INTERFACE I_State

PROPERTY Description : STRING
GET
END_GET
END_PROPERTY

METHOD ErrorDetected : BOOL
VAR_IN_OUT
	errorEvents		: ST_ErrorEvents;
END_VAR
END_METHOD

METHOD HeatIsRequested : BOOL
VAR_INPUT
END_VAR
END_METHOD

METHOD LimitValuesAreExceeded  : BOOL
VAR_INPUT
END_VAR
END_METHOD

PROPERTY Name : String
GET
END_GET
END_PROPERTY

PROPERTY State : E_State
GET
END_GET
END_PROPERTY

METHOD TargetTemperatureReached : BOOL
VAR_INPUT
END_VAR
END_METHOD

METHOD UserPressedConfirmationButton : BOOL
VAR_INPUT
END_VAR
END_METHOD

METHOD UserPressedSwitchOffButton : BOOL
VAR_INPUT
END_VAR
END_METHOD

METHOD UserPressedSwitchOnButton : BOOL
VAR_INPUT
END_VAR
END_METHOD

METHOD WaterHasCooledDown : BOOL
VAR_INPUT
END_VAR
END_METHOD

END_INTERFACE

(* stored: Version 1.1.0.1
   Itf I_State: Id {ebee4276-c4cf-4931-866b-4251da6de24d}
   Property Description: Id {09fe3b11-4466-4002-a19f-d7f98022308d}
   Get Get: Id {fb376b64-5463-4c2d-a1bb-8dc6a8df688f}
   Method ErrorDetected: Id {1fadc6df-44ce-4163-8a9d-0b84f9d6da56}
   Method HeatIsRequested: Id {bd7aa1f8-5748-4535-ba75-c3d1e68d26b3}
   Method LimitValuesAreExceeded: Id {00119294-6b09-4037-a5f2-bdd6e49bdada}
   Property Name: Id {185febd2-623d-4463-8457-cd856daf23b0}
   Get Get: Id {706e1d71-bb03-45f8-9d3a-58a361b141c0}
   Property State: Id {68cd257f-c6c4-44a4-9754-52e144c1f6ae}
   Get Get: Id {41d88164-af8d-49fe-af55-96517754930f}
   Method TargetTemperatureReached: Id {6137e0ac-cc2f-4194-abc8-c58d06d8efb2}
   Method UserPressedConfirmationButton: Id {b88189c9-53e3-4282-a4b8-58c626086e8a}
   Method UserPressedSwitchOffButton: Id {7f4f9871-0a9d-420a-9d6c-53cc58e2ab19}
   Method UserPressedSwitchOnButton: Id {d09cf28e-8c67-4e8c-b208-ac82badb61d6}
   Method WaterHasCooledDown: Id {e3917a29-80c1-4c55-b2b6-70e54206fcde} *)
